{attribute addProperty BoxType "KL1184"}
{attribute addProperty Id "Channel_1Channel_70B606D100Channel_2Channel_70B606D100Channel_3Channel_70B606D100Channel_4Channel_70B606D100"}
{attribute addProperty CRC "940274349"}
{attribute addProperty SizeInBites "0"}
{attribute addProperty SizeInBytes "0"}
TYPE KL1184_380B72AD :
STRUCT
	{attribute addProperty Name "Channel_1"}
	Channel_1 : Channel_70B606D1;
	{attribute addProperty Name "Channel_2"}
	Channel_2 : Channel_70B606D1;
	{attribute addProperty Name "Channel_3"}
	Channel_3 : Channel_70B606D1;
	{attribute addProperty Name "Channel_4"}
	Channel_4 : Channel_70B606D1;
END_STRUCT
END_TYPE

(* stored: Version 1.2.0.0, ProductVersion 3.1.4024.9
   DUT KL1184_380B72AD: Id {5ac9bf6b-d003-438a-a0d2-7e9292531792} *)
